INTERFACE I_MetadataVisitor

METHOD VisitMetadatum
VAR_INPUT
	VisitingMetadatum : I_Metadata;
END_VAR
END_METHOD

END_INTERFACE

(* stored: Version 1.1.0.1, ProductVersion 3.1.4024.12
   Itf I_MetadataVisitor: Id {b7b62421-6c3e-46c2-a5a8-344716c075d1}
   Method VisitMetadatum: Id {aed4f3e3-326f-4635-89c0-4cb529786257} *)
